Staubli VAL3: xppWriteBack.pgx

program xppWriteBack(string XsResponse (dimensions=1))
begin
  //
  //header begin
  // PROGRAM xppWriteBack()
  //
  // pgm writes text via TCP/IP to XPP client socket on CS8
  //
  // input parms:
  //    XsResponse = string passed from calling program
  //
  // output parms:
  //    none
  //
  // called from:  xppCmdHandler()
  //
  // initial release:  KN
  // Release 2:  KN
  //  changed functionality from CS8 host to CS8 client
  //  updated documentation
  //header end
  //
  sioXPPclient=XsResponse
end
